{attribute 'qualified_only}
PROGRAM COMM_UR10
VAR
	FB1: FB_MBReadRegs;
	
	// IP address & Port of ModBUS Server //
	ipAddr         					: STRING(15) := '192.168.1.13';
	iMBPort							: UINT := 502;
	
	// Function Blocks to extract robot information //
	// UR Robot Addresses and Array Sizes //
	nAddrrToolTCPCart				: WORD := 400;
	nAddrrToolTCPRot				: WORD := 403;
	nAddrrURAngles					: WORD := 270;
	nAddrrURAnglesVelocity			: WORD := 280;
	nAddrrURAnglesCurrent			: WORD := 290;
	nAddrrURAnglesTemp				: WORD := 300;
	nAddrrURJointMode				: WORD := 310;	
	nAddrrURState					: WORD := 260;
	nAddrrURProgAction				: WORD := 136;
	nAddrrURProgState				: WORD := 128;
	nAddrrPLCProgState				: WORD := 137;
	
	nQtyUnit						: WORD := 1;
	nQtyCart						: WORD := 3;
	nQtyRot							: WORD := 3;	
	nQtyURAxes						: WORD := 6;
		
	
	// Blocks //
	
	// Robot Angles information //	
	fbURAngles						: FB_MBReadRegs;
	// Robot Angles Velocity information //	
	fbURAnglesVelocity				: FB_MBReadRegs;
	// Robot Angles Current information //	
	fbURAnglesCurrent				: FB_MBReadRegs;
	// Robot Angles Temperature information //	
	fbURAnglesTemp					: FB_MBReadRegs;
	// Robot Joint Mode information //	
	fbURJointMode					: FB_MBReadRegs;
	// Robot Tool TCP Cart //	
	fbTool_TCP_Cartesian			: FB_MBReadRegs;
	// Robot Tool TCP Rot //
	fbTool_TCP_Rotation				: FB_MBReadRegs;
	// Robot Status //
	fbURRobot_Status				: FB_MBReadRegs;
	
	// Robot program start //
	fbURprogram_start				: FB_MBWriteRegs;
	// Robot state in program //
	fbUR_state_in_program			: FB_MBReadRegs;
	// PLC state in program //
	fbPLC_state_in_program			: FB_MBWriteRegs;
	
		
	// Reading Register - FB //
	fbReadRegs						: FB_MBReadRegs;
	bReadRegs						: BOOL;
	bReadRegsBusy   				: BOOL;
	bReadRegsError  				: BOOL;
	nReadRegsErrorId        		: UDINT;	
	
	// Writing Register - FB //
	fbWriteRegs						: FB_MBWriteRegs;
	bWriteRegs						: BOOL;
	bWriteRegsBusy   				: BOOL;
	bWriteRegsError  				: BOOL;
	nWriteRegsErrorId        		: UDINT;	
	
	// Error Variables //
	bError1, bError2, bError3		: BOOL;
	nErrID1, nErrID2, nErrID3		: UDINT;
	cbRead1, cbRead2, cbRead3		: UDINT;
	
	// Timers //
	TONreaders						: TON;
	TONwriters						: TON;
	tRefresh						: TIME := T#0.5S;
	tGiveUp							: TIME := T#2S;	
	
END_VAR

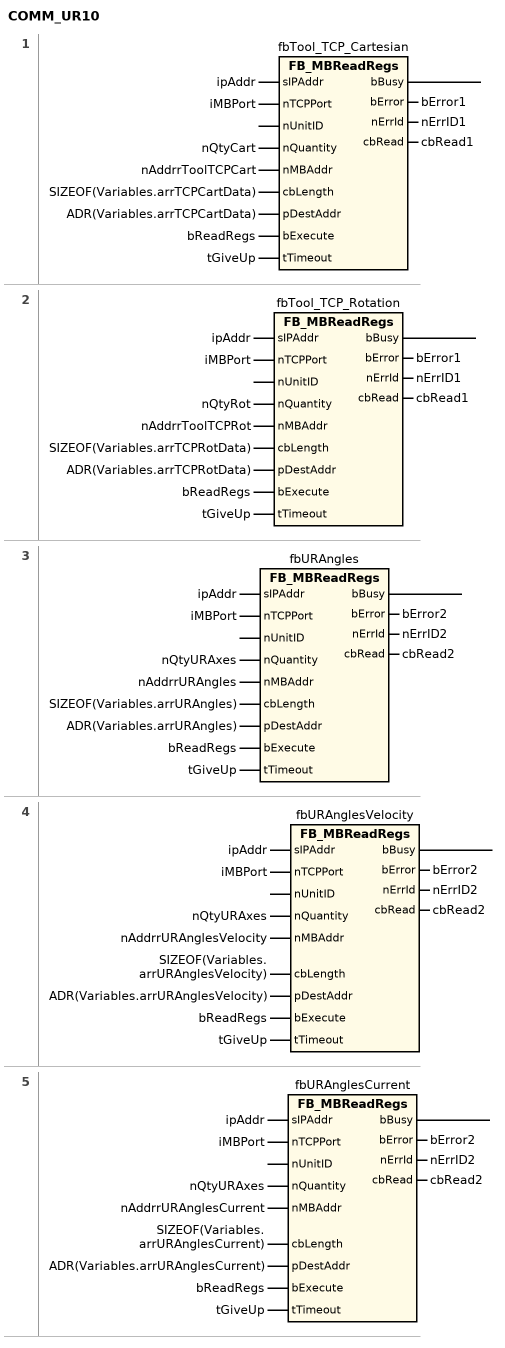
// NETWORK 1
fbTool_TCP_Cartesian(
    sIPAddr := ipAddr,
    nTCPPort := iMBPort,
    nQuantity := nQtyCart,
    nMBAddr := nAddrrToolTCPCart,
    cbLength := SIZEOF(Variables.arrTCPCartData),
    pDestAddr := ADR(Variables.arrTCPCartData),
    bExecute := bReadRegs,
    tTimeout := tGiveUp,
    bError => bError1,
    nErrId => nErrID1,
    cbRead => cbRead1); // FB_MBReadRegs

// NETWORK 2
fbTool_TCP_Rotation(
    sIPAddr := ipAddr,
    nTCPPort := iMBPort,
    nQuantity := nQtyRot,
    nMBAddr := nAddrrToolTCPRot,
    cbLength := SIZEOF(Variables.arrTCPRotData),
    pDestAddr := ADR(Variables.arrTCPRotData),
    bExecute := bReadRegs,
    tTimeout := tGiveUp,
    bError => bError1,
    nErrId => nErrID1,
    cbRead => cbRead1); // FB_MBReadRegs

// NETWORK 3
fbURAngles(
    sIPAddr := ipAddr,
    nTCPPort := iMBPort,
    nQuantity := nQtyURAxes,
    nMBAddr := nAddrrURAngles,
    cbLength := SIZEOF(Variables.arrURAngles),
    pDestAddr := ADR(Variables.arrURAngles),
    bExecute := bReadRegs,
    tTimeout := tGiveUp,
    bError => bError2,
    nErrId => nErrID2,
    cbRead => cbRead2); // FB_MBReadRegs

// NETWORK 4
fbURAnglesVelocity(
    sIPAddr := ipAddr,
    nTCPPort := iMBPort,
    nQuantity := nQtyURAxes,
    nMBAddr := nAddrrURAnglesVelocity,
    cbLength := SIZEOF(Variables.arrURAnglesVelocity),
    pDestAddr := ADR(Variables.arrURAnglesVelocity),
    bExecute := bReadRegs,
    tTimeout := tGiveUp,
    bError => bError2,
    nErrId => nErrID2,
    cbRead => cbRead2); // FB_MBReadRegs

// NETWORK 5
fbURAnglesCurrent(
    sIPAddr := ipAddr,
    nTCPPort := iMBPort,
    nQuantity := nQtyURAxes,
    nMBAddr := nAddrrURAnglesCurrent,
    cbLength := SIZEOF(Variables.arrURAnglesCurrent),
    pDestAddr := ADR(Variables.arrURAnglesCurrent),
    bExecute := bReadRegs,
    tTimeout := tGiveUp,
    bError => bError2,
    nErrId => nErrID2,
    cbRead => cbRead2); // FB_MBReadRegs

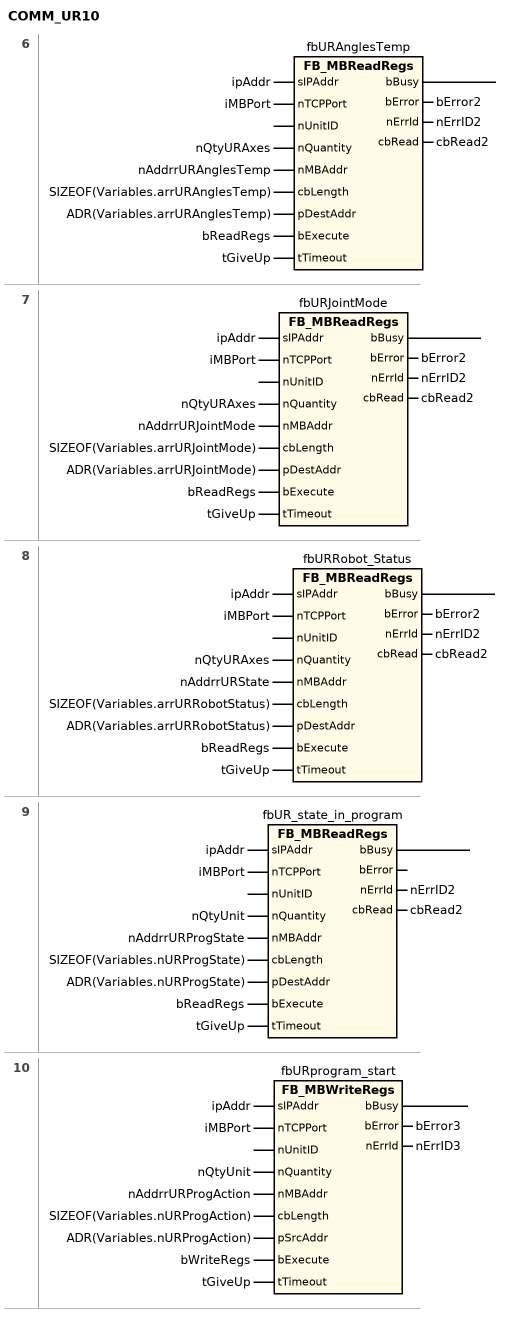
// NETWORK 6
fbURAnglesTemp(
    sIPAddr := ipAddr,
    nTCPPort := iMBPort,
    nQuantity := nQtyURAxes,
    nMBAddr := nAddrrURAnglesTemp,
    cbLength := SIZEOF(Variables.arrURAnglesTemp),
    pDestAddr := ADR(Variables.arrURAnglesTemp),
    bExecute := bReadRegs,
    tTimeout := tGiveUp,
    bError => bError2,
    nErrId => nErrID2,
    cbRead => cbRead2); // FB_MBReadRegs

// NETWORK 7
fbURJointMode(
    sIPAddr := ipAddr,
    nTCPPort := iMBPort,
    nQuantity := nQtyURAxes,
    nMBAddr := nAddrrURJointMode,
    cbLength := SIZEOF(Variables.arrURJointMode),
    pDestAddr := ADR(Variables.arrURJointMode),
    bExecute := bReadRegs,
    tTimeout := tGiveUp,
    bError => bError2,
    nErrId => nErrID2,
    cbRead => cbRead2); // FB_MBReadRegs

// NETWORK 8
fbURRobot_Status(
    sIPAddr := ipAddr,
    nTCPPort := iMBPort,
    nQuantity := nQtyURAxes,
    nMBAddr := nAddrrURState,
    cbLength := SIZEOF(Variables.arrURRobotStatus),
    pDestAddr := ADR(Variables.arrURRobotStatus),
    bExecute := bReadRegs,
    tTimeout := tGiveUp,
    bError => bError2,
    nErrId => nErrID2,
    cbRead => cbRead2); // FB_MBReadRegs

// NETWORK 9
fbUR_state_in_program(
    sIPAddr := ipAddr,
    nTCPPort := iMBPort,
    nQuantity := nQtyUnit,
    nMBAddr := nAddrrURProgState,
    cbLength := SIZEOF(Variables.nURProgState),
    pDestAddr := ADR(Variables.nURProgState),
    bExecute := bReadRegs,
    tTimeout := tGiveUp,
    nErrId => nErrID2,
    cbRead => cbRead2); // FB_MBReadRegs

// NETWORK 10
fbURprogram_start(
    sIPAddr := ipAddr,
    nTCPPort := iMBPort,
    nQuantity := nQtyUnit,
    nMBAddr := nAddrrURProgAction,
    cbLength := SIZEOF(Variables.nURProgAction),
    pSrcAddr := ADR(Variables.nURProgAction),
    bExecute := bWriteRegs,
    tTimeout := tGiveUp,
    bError => bError3,
    nErrId => nErrID3); // FB_MBWriteRegs

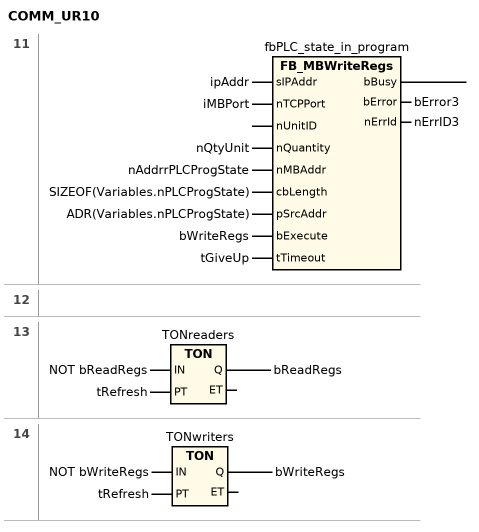
// NETWORK 11
fbPLC_state_in_program(
    sIPAddr := ipAddr,
    nTCPPort := iMBPort,
    nQuantity := nQtyUnit,
    nMBAddr := nAddrrPLCProgState,
    cbLength := SIZEOF(Variables.nPLCProgState),
    pSrcAddr := ADR(Variables.nPLCProgState),
    bExecute := bWriteRegs,
    tTimeout := tGiveUp,
    bError => bError3,
    nErrId => nErrID3); // FB_MBWriteRegs

// NETWORK 12

// NETWORK 13
TONreaders(IN := NOT bReadRegs, PT := tRefresh); // TON
bReadRegs := TONreaders.Q;

// NETWORK 14
TONwriters(IN := NOT bWriteRegs, PT := tRefresh); // TON
bWriteRegs := TONwriters.Q;

END_PROGRAM

(* stored: Version 1.1.0.1, ProductVersion 3.1.4024.0
   POU COMM_UR10: Id {6c3ee355-86ab-4b32-bb51-9ae35bb35eea}, SpecialFunc None *)
